INTERFACE I_BacklashCompensation

(*
    Handle positive/negative backlash compensation
    User needs to set the direction of backlash from the sign of the compensation value
    Backlash compensation is disabled during referencing (homing).
    When direction is positive/negative, further movement in the negative/positive direction not compensated
    further movement in the negative/positive direction will be compensated
*)
METHOD BacklashCompensation
VAR_INPUT
    Enable     : BOOL;
	Execute		: BOOL;
    Compensation	: LREAL;
    fRampVelocity	: LREAL := 10.0;
    DisableMode	: E_DISABLEMODE := E_DISABLEMODE.DisableModeHold;
END_VAR
END_METHOD

PROPERTY BacklashCompensationError : BOOL
GET
END_GET
END_PROPERTY

PROPERTY BacklashCompensationErrorID : UDINT
GET
END_GET
END_PROPERTY

PROPERTY DisableMode : E_DISABLEMODE
GET
END_GET
SET
END_SET
END_PROPERTY

PROPERTY Enable : BOOL
GET
END_GET
SET
END_SET
END_PROPERTY

PROPERTY MeasureBacklash : LREAL
GET
END_GET
END_PROPERTY

PROPERTY RampVelocity : LREAL
GET
END_GET
SET
END_SET
END_PROPERTY

PROPERTY Status : BOOL
GET
END_GET
END_PROPERTY

PROPERTY TargetCompensation : LREAL
GET
END_GET
SET
END_SET
END_PROPERTY

END_INTERFACE

(* stored: Version 1.1.0.1
   Itf I_BacklashCompensation: Id {c0dc76c5-ea53-4a27-aade-dbf12ab6b44d}
   Method BacklashCompensation: Id {8dc8359f-12ee-498a-aa0e-4230cfa1b09f}
   Property BacklashCompensationError: Id {6f1b59b6-4b74-42e0-b9fe-ffa15d3f45e7}
   Get Get: Id {daae0576-b11a-47a6-b8ad-fd2ba8bffdd8}
   Property BacklashCompensationErrorID: Id {401b0c6b-f002-4c91-8190-9716c225529b}
   Get Get: Id {11af064e-4fdb-4269-bde7-aa834e9e2b95}
   Property DisableMode: Id {0895cb27-228d-442d-be60-7b108cb8779a}
   Get Get: Id {5b639a65-3a92-4bfc-9bf1-017768c44834}
   Set Set: Id {0aaace7d-e7af-4d3a-8855-1d6a7fd1bbb2}
   Property Enable: Id {705e6fa8-d6ff-4042-8fed-7aa14453215a}
   Get Get: Id {d222f11b-678d-4c52-af6d-690095d252fa}
   Set Set: Id {d967ab92-050d-4b6e-a67c-f99f28890f47}
   Property MeasureBacklash: Id {ff081112-3182-493d-846e-c2192c5f77d6}
   Get Get: Id {5dbd065d-c6db-421a-8993-7aa4f3a00024}
   Property RampVelocity: Id {8cd265dd-6c90-4161-ac4a-ff52460744b4}
   Get Get: Id {4f1c0d40-5241-4737-91fd-a99f6c34c0fc}
   Set Set: Id {499ddcbb-00a7-4cff-8d4b-d6041629a57c}
   Property Status: Id {ad5dd29e-09ce-4214-902d-59b991e685e4}
   Get Get: Id {a39149e1-eecc-44bb-bc32-b9385b7fdf09}
   Property TargetCompensation: Id {84e0b4a7-d241-4df9-a3cd-164122514251}
   Get Get: Id {636b5cc6-bb68-4499-971f-12fd2d4192c7}
   Set Set: Id {9da4ffef-d58b-4b0d-9640-614faf3010c2} *)
